PROGRAM OP160_MASTER4_IO
VAR
	OP160_MAS4_PORT1_BYTE1_DI_MODULE_1 AT %I* : BYTE;
	OP160_MAS4_PORT1_BYTE2_DI_MODULE_1 AT %I* : BYTE;
	OP160_MAS4_PORT2_BYTE1_DI_MODULE_2 AT %I* : BYTE;
	OP160_MAS4_PORT2_BYTE2_DI_MODULE_2 AT %I* : BYTE;
	OP160_MAS4_PORT3_BYTE1_DI_MODULE_3 AT %I* : BYTE;
	OP160_MAS4_PORT3_BYTE2_DI_MODULE_3 AT %I* : BYTE;
	OP160_MAS4_PORT4_BYTE1_DI_MODULE_4 AT %I* : BYTE;
	OP160_MAS4_PORT4_BYTE2_DI_MODULE_4 AT %I* : BYTE;
	
	OP160_MAS4_PORT5_BYTE1_DO_MODULE_1 AT %Q* : BYTE;
	OP160_MAS4_PORT5_BYTE2_DO_MODULE_1 AT %Q* : BYTE;
	OP160_MAS4_PORT5_BYTE3_DO_MODULE_1 AT %Q* : BYTE;
	OP160_MAS4_PORT5_BYTE4_DO_MODULE_1 AT %Q* : BYTE;
	OP160_MAS4_PORT6_BYTE1_DO_MODULE_2 AT %Q* : BYTE;
	OP160_MAS4_PORT6_BYTE2_DO_MODULE_2 AT %Q* : BYTE;
	OP160_MAS4_PORT6_BYTE3_DO_MODULE_2 AT %Q* : BYTE;
	OP160_MAS4_PORT6_BYTE4_DO_MODULE_2 AT %Q* : BYTE;
	
	
	

	BYTE_AS_BIT_0: BYTE_AS_BIT;
	BYTE_AS_BIT_1: BYTE_AS_BIT;
	BYTE_AS_BIT_2: BYTE_AS_BIT;
	BYTE_AS_BIT_3: BYTE_AS_BIT;
	BYTE_AS_BIT_4: BYTE_AS_BIT;
	BYTE_AS_BIT_5: BYTE_AS_BIT;
	BYTE_AS_BIT_6: BYTE_AS_BIT;
	BYTE_AS_BIT_7: BYTE_AS_BIT;
	
		
	BIT_AS_BYTE_0: BIT_AS_BYTE;
	BIT_AS_BYTE_1: BIT_AS_BYTE;
	BIT_AS_BYTE_2: BIT_AS_BYTE;
	BIT_AS_BYTE_3: BIT_AS_BYTE;
	BIT_AS_BYTE_4: BIT_AS_BYTE;
	BIT_AS_BYTE_5: BIT_AS_BYTE;
	BIT_AS_BYTE_6: BIT_AS_BYTE;
	BIT_AS_BYTE_7: BIT_AS_BYTE;
END_VAR

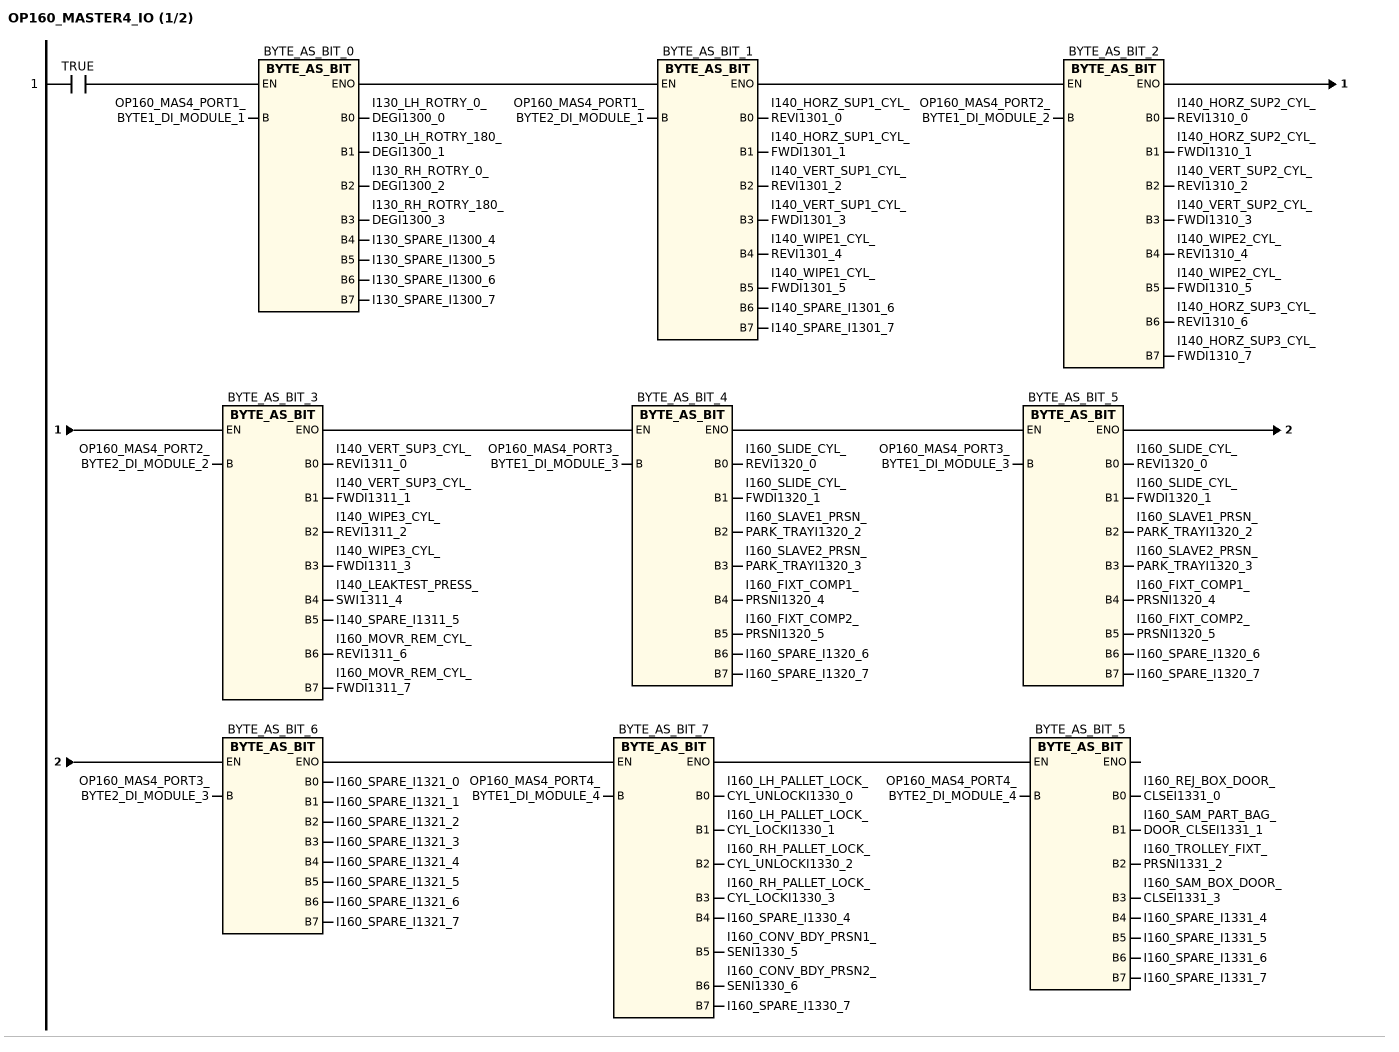
// NETWORK 1
BYTE_AS_BIT_0(
    B := OP160_MAS4_PORT1_BYTE1_DI_MODULE_1,
    B0 => I130_LH_ROTRY_0_DEGI1300_0,
    B1 => I130_LH_ROTRY_180_DEGI1300_1,
    B2 => I130_RH_ROTRY_0_DEGI1300_2,
    B3 => I130_RH_ROTRY_180_DEGI1300_3,
    B4 => I130_SPARE_I1300_4,
    B5 => I130_SPARE_I1300_5,
    B6 => I130_SPARE_I1300_6,
    B7 => I130_SPARE_I1300_7); // BYTE_AS_BIT
BYTE_AS_BIT_1(
    B := OP160_MAS4_PORT1_BYTE2_DI_MODULE_1,
    B0 => I140_HORZ_SUP1_CYL_REVI1301_0,
    B1 => I140_HORZ_SUP1_CYL_FWDI1301_1,
    B2 => I140_VERT_SUP1_CYL_REVI1301_2,
    B3 => I140_VERT_SUP1_CYL_FWDI1301_3,
    B4 => I140_WIPE1_CYL_REVI1301_4,
    B5 => I140_WIPE1_CYL_FWDI1301_5,
    B6 => I140_SPARE_I1301_6,
    B7 => I140_SPARE_I1301_7); // BYTE_AS_BIT
BYTE_AS_BIT_2(
    B := OP160_MAS4_PORT2_BYTE1_DI_MODULE_2,
    B0 => I140_HORZ_SUP2_CYL_REVI1310_0,
    B1 => I140_HORZ_SUP2_CYL_FWDI1310_1,
    B2 => I140_VERT_SUP2_CYL_REVI1310_2,
    B3 => I140_VERT_SUP2_CYL_FWDI1310_3,
    B4 => I140_WIPE2_CYL_REVI1310_4,
    B5 => I140_WIPE2_CYL_FWDI1310_5,
    B6 => I140_HORZ_SUP3_CYL_REVI1310_6,
    B7 => I140_HORZ_SUP3_CYL_FWDI1310_7); // BYTE_AS_BIT
BYTE_AS_BIT_3(
    B := OP160_MAS4_PORT2_BYTE2_DI_MODULE_2,
    B0 => I140_VERT_SUP3_CYL_REVI1311_0,
    B1 => I140_VERT_SUP3_CYL_FWDI1311_1,
    B2 => I140_WIPE3_CYL_REVI1311_2,
    B3 => I140_WIPE3_CYL_FWDI1311_3,
    B4 => I140_LEAKTEST_PRESS_SWI1311_4,
    B5 => I140_SPARE_I1311_5,
    B6 => I160_MOVR_REM_CYL_REVI1311_6,
    B7 => I160_MOVR_REM_CYL_FWDI1311_7); // BYTE_AS_BIT
BYTE_AS_BIT_4(
    B := OP160_MAS4_PORT3_BYTE1_DI_MODULE_3,
    B0 => I160_SLIDE_CYL_REVI1320_0,
    B1 => I160_SLIDE_CYL_FWDI1320_1,
    B2 => I160_SLAVE1_PRSN_PARK_TRAYI1320_2,
    B3 => I160_SLAVE2_PRSN_PARK_TRAYI1320_3,
    B4 => I160_FIXT_COMP1_PRSNI1320_4,
    B5 => I160_FIXT_COMP2_PRSNI1320_5,
    B6 => I160_SPARE_I1320_6,
    B7 => I160_SPARE_I1320_7); // BYTE_AS_BIT
BYTE_AS_BIT_5(
    B := OP160_MAS4_PORT3_BYTE1_DI_MODULE_3,
    B0 => I160_SLIDE_CYL_REVI1320_0,
    B1 => I160_SLIDE_CYL_FWDI1320_1,
    B2 => I160_SLAVE1_PRSN_PARK_TRAYI1320_2,
    B3 => I160_SLAVE2_PRSN_PARK_TRAYI1320_3,
    B4 => I160_FIXT_COMP1_PRSNI1320_4,
    B5 => I160_FIXT_COMP2_PRSNI1320_5,
    B6 => I160_SPARE_I1320_6,
    B7 => I160_SPARE_I1320_7); // BYTE_AS_BIT
BYTE_AS_BIT_6(
    B := OP160_MAS4_PORT3_BYTE2_DI_MODULE_3,
    B0 => I160_SPARE_I1321_0,
    B1 => I160_SPARE_I1321_1,
    B2 => I160_SPARE_I1321_2,
    B3 => I160_SPARE_I1321_3,
    B4 => I160_SPARE_I1321_4,
    B5 => I160_SPARE_I1321_5,
    B6 => I160_SPARE_I1321_6,
    B7 => I160_SPARE_I1321_7); // BYTE_AS_BIT
BYTE_AS_BIT_7(
    B := OP160_MAS4_PORT4_BYTE1_DI_MODULE_4,
    B0 => I160_LH_PALLET_LOCK_CYL_UNLOCKI1330_0,
    B1 => I160_LH_PALLET_LOCK_CYL_LOCKI1330_1,
    B2 => I160_RH_PALLET_LOCK_CYL_UNLOCKI1330_2,
    B3 => I160_RH_PALLET_LOCK_CYL_LOCKI1330_3,
    B4 => I160_SPARE_I1330_4,
    B5 => I160_CONV_BDY_PRSN1_SENI1330_5,
    B6 => I160_CONV_BDY_PRSN2_SENI1330_6,
    B7 => I160_SPARE_I1330_7); // BYTE_AS_BIT
BYTE_AS_BIT_5(
    B := OP160_MAS4_PORT4_BYTE2_DI_MODULE_4,
    B0 => I160_REJ_BOX_DOOR_CLSEI1331_0,
    B1 => I160_SAM_PART_BAG_DOOR_CLSEI1331_1,
    B2 => I160_TROLLEY_FIXT_PRSNI1331_2,
    B3 => I160_SAM_BOX_DOOR_CLSEI1331_3,
    B4 => I160_SPARE_I1331_4,
    B5 => I160_SPARE_I1331_5,
    B6 => I160_SPARE_I1331_6,
    B7 => I160_SPARE_I1331_7); // BYTE_AS_BIT

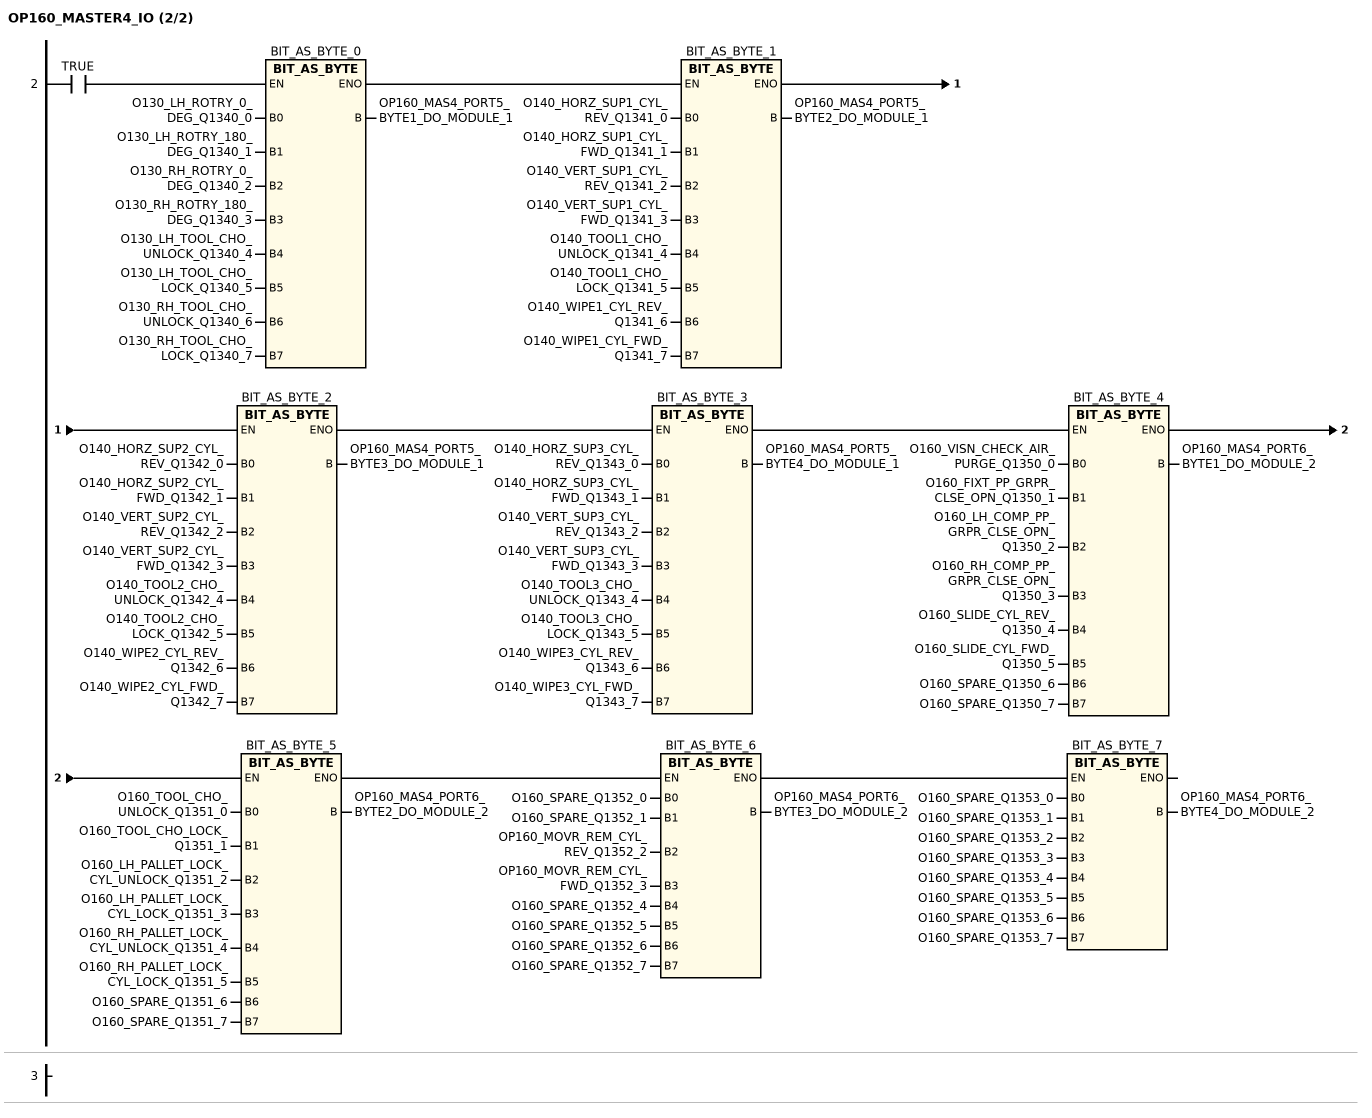
// NETWORK 2
BIT_AS_BYTE_0(
    B0 := O130_LH_ROTRY_0_DEG_Q1340_0,
    B1 := O130_LH_ROTRY_180_DEG_Q1340_1,
    B2 := O130_RH_ROTRY_0_DEG_Q1340_2,
    B3 := O130_RH_ROTRY_180_DEG_Q1340_3,
    B4 := O130_LH_TOOL_CHO_UNLOCK_Q1340_4,
    B5 := O130_LH_TOOL_CHO_LOCK_Q1340_5,
    B6 := O130_RH_TOOL_CHO_UNLOCK_Q1340_6,
    B7 := O130_RH_TOOL_CHO_LOCK_Q1340_7,
    B => OP160_MAS4_PORT5_BYTE1_DO_MODULE_1); // BIT_AS_BYTE
BIT_AS_BYTE_1(
    B0 := O140_HORZ_SUP1_CYL_REV_Q1341_0,
    B1 := O140_HORZ_SUP1_CYL_FWD_Q1341_1,
    B2 := O140_VERT_SUP1_CYL_REV_Q1341_2,
    B3 := O140_VERT_SUP1_CYL_FWD_Q1341_3,
    B4 := O140_TOOL1_CHO_UNLOCK_Q1341_4,
    B5 := O140_TOOL1_CHO_LOCK_Q1341_5,
    B6 := O140_WIPE1_CYL_REV_Q1341_6,
    B7 := O140_WIPE1_CYL_FWD_Q1341_7,
    B => OP160_MAS4_PORT5_BYTE2_DO_MODULE_1); // BIT_AS_BYTE
BIT_AS_BYTE_2(
    B0 := O140_HORZ_SUP2_CYL_REV_Q1342_0,
    B1 := O140_HORZ_SUP2_CYL_FWD_Q1342_1,
    B2 := O140_VERT_SUP2_CYL_REV_Q1342_2,
    B3 := O140_VERT_SUP2_CYL_FWD_Q1342_3,
    B4 := O140_TOOL2_CHO_UNLOCK_Q1342_4,
    B5 := O140_TOOL2_CHO_LOCK_Q1342_5,
    B6 := O140_WIPE2_CYL_REV_Q1342_6,
    B7 := O140_WIPE2_CYL_FWD_Q1342_7,
    B => OP160_MAS4_PORT5_BYTE3_DO_MODULE_1); // BIT_AS_BYTE
BIT_AS_BYTE_3(
    B0 := O140_HORZ_SUP3_CYL_REV_Q1343_0,
    B1 := O140_HORZ_SUP3_CYL_FWD_Q1343_1,
    B2 := O140_VERT_SUP3_CYL_REV_Q1343_2,
    B3 := O140_VERT_SUP3_CYL_FWD_Q1343_3,
    B4 := O140_TOOL3_CHO_UNLOCK_Q1343_4,
    B5 := O140_TOOL3_CHO_LOCK_Q1343_5,
    B6 := O140_WIPE3_CYL_REV_Q1343_6,
    B7 := O140_WIPE3_CYL_FWD_Q1343_7,
    B => OP160_MAS4_PORT5_BYTE4_DO_MODULE_1); // BIT_AS_BYTE
BIT_AS_BYTE_4(
    B0 := O160_VISN_CHECK_AIR_PURGE_Q1350_0,
    B1 := O160_FIXT_PP_GRPR_CLSE_OPN_Q1350_1,
    B2 := O160_LH_COMP_PP_GRPR_CLSE_OPN_Q1350_2,
    B3 := O160_RH_COMP_PP_GRPR_CLSE_OPN_Q1350_3,
    B4 := O160_SLIDE_CYL_REV_Q1350_4,
    B5 := O160_SLIDE_CYL_FWD_Q1350_5,
    B6 := O160_SPARE_Q1350_6,
    B7 := O160_SPARE_Q1350_7,
    B => OP160_MAS4_PORT6_BYTE1_DO_MODULE_2); // BIT_AS_BYTE
BIT_AS_BYTE_5(
    B0 := O160_TOOL_CHO_UNLOCK_Q1351_0,
    B1 := O160_TOOL_CHO_LOCK_Q1351_1,
    B2 := O160_LH_PALLET_LOCK_CYL_UNLOCK_Q1351_2,
    B3 := O160_LH_PALLET_LOCK_CYL_LOCK_Q1351_3,
    B4 := O160_RH_PALLET_LOCK_CYL_UNLOCK_Q1351_4,
    B5 := O160_RH_PALLET_LOCK_CYL_LOCK_Q1351_5,
    B6 := O160_SPARE_Q1351_6,
    B7 := O160_SPARE_Q1351_7,
    B => OP160_MAS4_PORT6_BYTE2_DO_MODULE_2); // BIT_AS_BYTE
BIT_AS_BYTE_6(
    B0 := O160_SPARE_Q1352_0,
    B1 := O160_SPARE_Q1352_1,
    B2 := OP160_MOVR_REM_CYL_REV_Q1352_2,
    B3 := OP160_MOVR_REM_CYL_FWD_Q1352_3,
    B4 := O160_SPARE_Q1352_4,
    B5 := O160_SPARE_Q1352_5,
    B6 := O160_SPARE_Q1352_6,
    B7 := O160_SPARE_Q1352_7,
    B => OP160_MAS4_PORT6_BYTE3_DO_MODULE_2); // BIT_AS_BYTE
BIT_AS_BYTE_7(
    B0 := O160_SPARE_Q1353_0,
    B1 := O160_SPARE_Q1353_1,
    B2 := O160_SPARE_Q1353_2,
    B3 := O160_SPARE_Q1353_3,
    B4 := O160_SPARE_Q1353_4,
    B5 := O160_SPARE_Q1353_5,
    B6 := O160_SPARE_Q1353_6,
    B7 := O160_SPARE_Q1353_7,
    B => OP160_MAS4_PORT6_BYTE4_DO_MODULE_2); // BIT_AS_BYTE

// NETWORK 3

END_PROGRAM

(* stored: Version 1.1.0.1, ProductVersion 3.1.4024.11
   POU OP160_MASTER4_IO: Id {cb9c578b-ba92-47ec-9483-759cee649640}, SpecialFunc None *)
